INTERFACE I_Request EXTENDS I_Disposable

PROPERTY PUBLIC CreatedTimestamp : I_Timestamp
GET
END_GET
END_PROPERTY

PROPERTY PUBLIC Header : I_RequestHeader
GET
END_GET
END_PROPERTY

PROPERTY PUBLIC Payload : REFERENCE TO STRING(Constants.REQUEST_PAYLOAD_STRING_SIZE);
GET
END_GET
END_PROPERTY

END_INTERFACE

(* stored: Version 1.1.0.1, ProductVersion 3.1.4024.12
   Itf I_Request: Id {09fb0484-0921-4add-a143-8e5b5a4ec79b}
   Property CreatedTimestamp: Id {6654dbac-bbdc-4e29-abd7-f7bae031a16b}
   Get Get: Id {a8827976-4218-49a8-958a-254625df3344}
   Property Header: Id {e48d46f2-b1ae-4764-81c7-c961d7cf6a85}
   Get Get: Id {aa2814e0-af57-4ffe-a8c4-7e1da4004afd}
   Property Payload: Id {9009cd02-59c3-442d-b694-7fd07046c812}
   Get Get: Id {a4712b06-3c0b-406d-a560-cb95d77529be} *)
